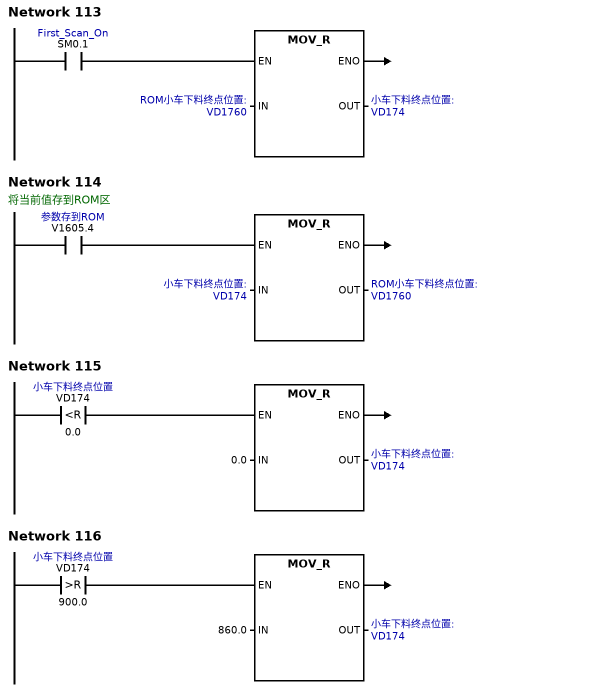
[picture p72: SBR20 networks 113-116]
Network 113
LD     First_Scan_On:SM0.1
MOVR   ROM小车下料终点位置:VD1760, 小车下料终点位置:VD174
Network 114
// 将当前值存到ROM区
LD     参数存到ROM:V1605.4
MOVR   小车下料终点位置:VD174, ROM小车下料终点位置:VD1760
Network 115
LDR<   小车下料终点位置:VD174, 0.0
MOVR   0.0, 小车下料终点位置:VD174
Network 116
LDR>   小车下料终点位置:VD174, 900.0
MOVR   860.0, 小车下料终点位置:VD174
END_SUBROUTINE_BLOCK

SUBROUTINE_BLOCK 故障报警:SBR21
TITLE=子程序注释
BEGIN
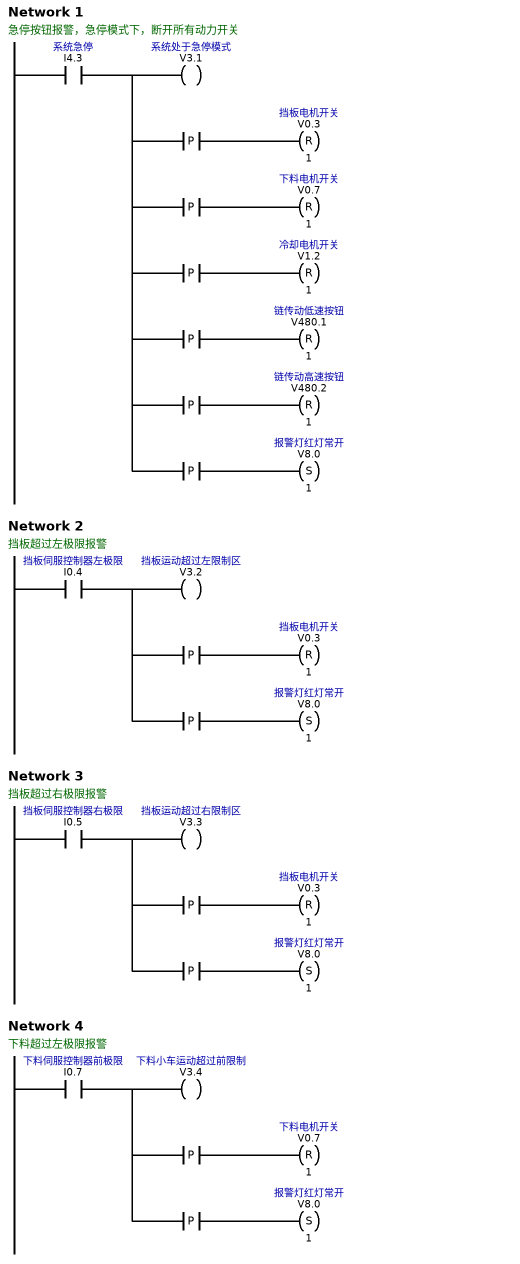
Network 1
// 急停按钮报警，急停模式下，断开所有动力开关
LD     系统急停:I4.3
LPS
=      系统处于急停模式:V3.1
EU
R      挡板电机开关:V0.3, 1
LRD
EU
R      下料电机开关:V0.7, 1
LRD
EU
R      冷却电机开关:V1.2, 1
LRD
EU
R      链传动低速按钮:V480.1, 1
LRD
EU
R      链传动高速按钮:V480.2, 1
LPP
EU
S      报警灯红灯常开:V8.0, 1
Network 2
// 挡板超过左极限报警
LD     挡板伺服控制器左极限:I0.4
LPS
=      挡板运动超过左限制区:V3.2
EU
R      挡板电机开关:V0.3, 1
LPP
EU
S      报警灯红灯常开:V8.0, 1
Network 3
// 挡板超过右极限报警
LD     挡板伺服控制器右极限:I0.5
LPS
=      挡板运动超过右限制区:V3.3
EU
R      挡板电机开关:V0.3, 1
LPP
EU
S      报警灯红灯常开:V8.0, 1
Network 4
// 下料超过左极限报警
LD     下料伺服控制器前极限:I0.7
LPS
=      下料小车运动超过前限制:V3.4
EU
R      下料电机开关:V0.7, 1
LPP
EU
S      报警灯红灯常开:V8.0, 1
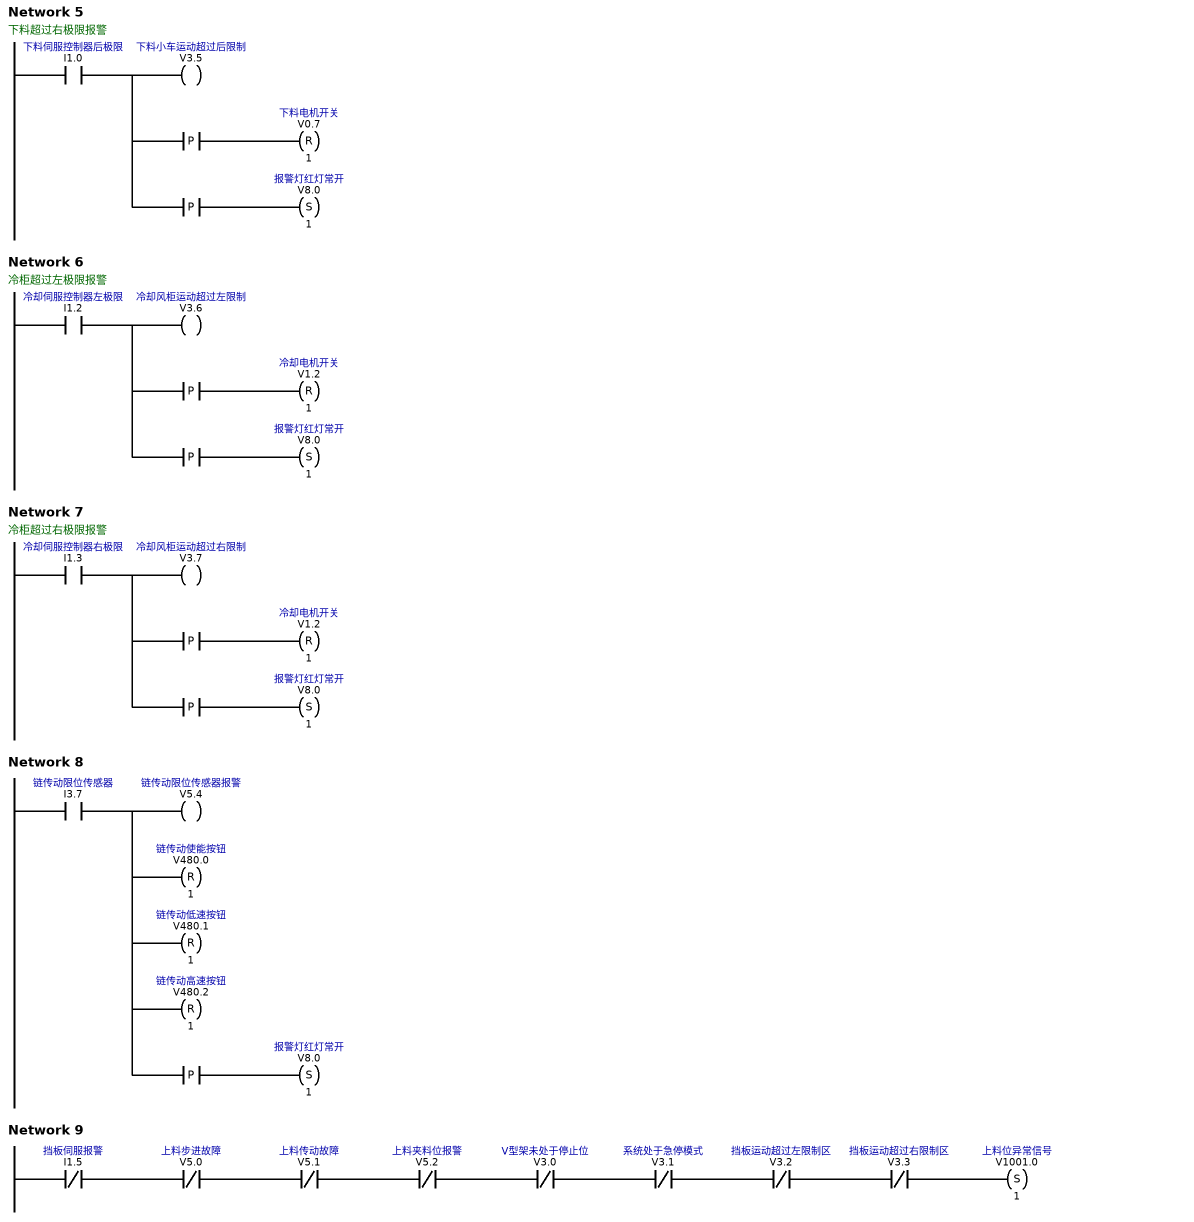
Network 5
// 下料超过右极限报警
LD     下料伺服控制器后极限:I1.0
LPS
=      下料小车运动超过后限制:V3.5
EU
R      下料电机开关:V0.7, 1
LPP
EU
S      报警灯红灯常开:V8.0, 1
Network 6
// 冷柜超过左极限报警
LD     冷却伺服控制器左极限:I1.2
LPS
=      冷却风柜运动超过左限制:V3.6
EU
R      冷却电机开关:V1.2, 1
LPP
EU
S      报警灯红灯常开:V8.0, 1
Network 7
// 冷柜超过右极限报警
LD     冷却伺服控制器右极限:I1.3
LPS
=      冷却风柜运动超过右限制:V3.7
EU
R      冷却电机开关:V1.2, 1
LPP
EU
S      报警灯红灯常开:V8.0, 1
Network 8
LD     链传动限位传感器:I3.7
=      链传动限位传感器报警:V5.4
R      链传动使能按钮:V480.0, 1
R      链传动低速按钮:V480.1, 1
R      链传动高速按钮:V480.2, 1
EU
S      报警灯红灯常开:V8.0, 1
Network 9
LDN    挡板伺服报警:I1.5
AN     上料步进故障:V5.0
AN     上料传动故障:V5.1
AN     上料夹料位报警:V5.2
AN     V型架未处于停止位:V3.0
AN     系统处于急停模式:V3.1
AN     挡板运动超过左限制区:V3.2
AN     挡板运动超过右限制区:V3.3
S      上料位异常信号:V1001.0, 1
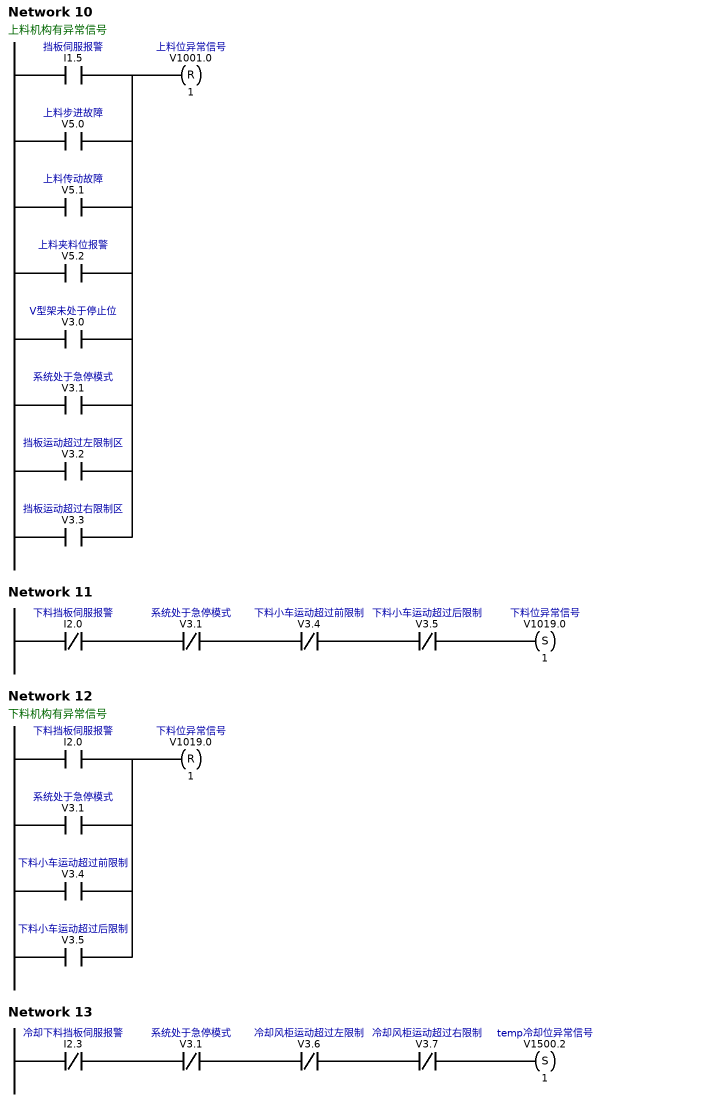
Network 10
// 上料机构有异常信号
LD     挡板伺服报警:I1.5
O      上料步进故障:V5.0
O      上料传动故障:V5.1
O      上料夹料位报警:V5.2
O      V型架未处于停止位:V3.0
O      系统处于急停模式:V3.1
O      挡板运动超过左限制区:V3.2
O      挡板运动超过右限制区:V3.3
R      上料位异常信号:V1001.0, 1
Network 11
LDN    下料挡板伺服报警:I2.0
AN     系统处于急停模式:V3.1
AN     下料小车运动超过前限制:V3.4
AN     下料小车运动超过后限制:V3.5
S      下料位异常信号:V1019.0, 1
Network 12
// 下料机构有异常信号
LD     下料挡板伺服报警:I2.0
O      系统处于急停模式:V3.1
O      下料小车运动超过前限制:V3.4
O      下料小车运动超过后限制:V3.5
R      下料位异常信号:V1019.0, 1
Network 13
LDN    冷却下料挡板伺服报警:I2.3
AN     系统处于急停模式:V3.1
AN     冷却风柜运动超过左限制:V3.6
AN     冷却风柜运动超过右限制:V3.7
S      temp冷却位异常信号:V1500.2, 1
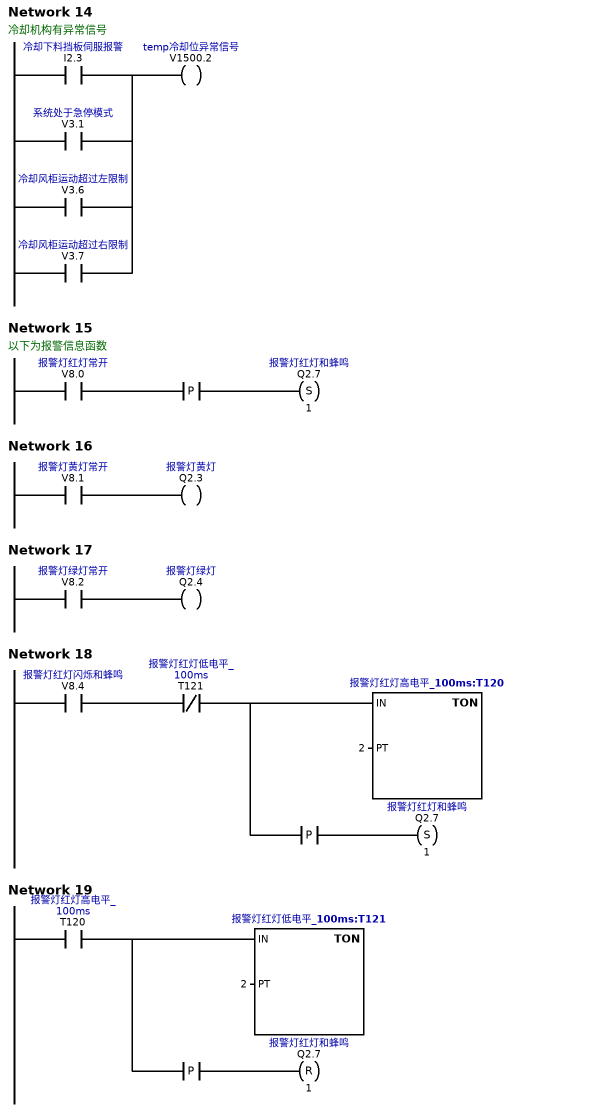
Network 14
// 冷却机构有异常信号
LD     冷却下料挡板伺服报警:I2.3
O      系统处于急停模式:V3.1
O      冷却风柜运动超过左限制:V3.6
O      冷却风柜运动超过右限制:V3.7
=      temp冷却位异常信号:V1500.2
Network 15
// 以下为报警信息函数
LD     报警灯红灯常开:V8.0
EU
S      报警灯红灯和蜂鸣:Q2.7, 1
Network 16
LD     报警灯黄灯常开:V8.1
=      报警灯黄灯:Q2.3
Network 17
LD     报警灯绿灯常开:V8.2
=      报警灯绿灯:Q2.4
Network 18
LD     报警灯红灯闪烁和蜂鸣:V8.4
AN     报警灯红灯低电平_100ms:T121
TON    报警灯红灯高电平_100ms:T120, 2
EU
S      报警灯红灯和蜂鸣:Q2.7, 1
Network 19
LD     报警灯红灯高电平_100ms:T120
TON    报警灯红灯低电平_100ms:T121, 2
EU
R      报警灯红灯和蜂鸣:Q2.7, 1
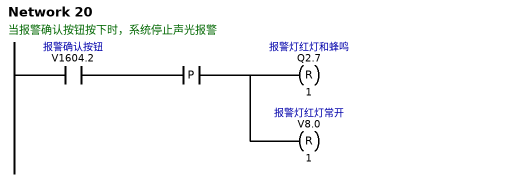
Network 20
// 当报警确认按钮按下时，系统停止声光报警
LD     报警确认按钮:V1604.2
EU
R      报警灯红灯和蜂鸣:Q2.7, 1
R      报警灯红灯常开:V8.0, 1
END_SUBROUTINE_BLOCK

SUBROUTINE_BLOCK 总控机监控部分程序:SBR22
TITLE=子程序注释
BEGIN
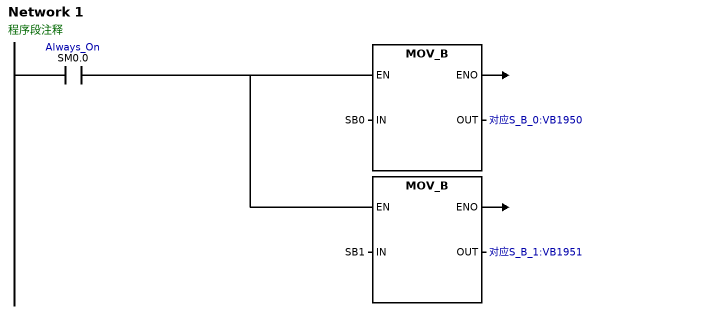
Network 1
// 程序段注释
// (network saved uncompiled; LAD cells follow)
// row 0: c0 -| |- Always_On:SM0.0  c1 -- v  c2 --  c3 [MOV_B EN:=power@row0, IN:=SB0, ENO=>power, OUT=>对应S_B_0:VB1950]  c4 ->
// row 1: c1 ^v  c3 [box]
// row 2: c1 ^  c2 --  c3 [MOV_B EN:=power@row2, IN:=SB1, ENO=>power, OUT=>对应S_B_1:VB1951]  c4 ->
// row 3: c3 [box]
END_SUBROUTINE_BLOCK
